{attribute 'GeneratedUsingTerminal: EPP1322-0001-0017'}
{attribute addProperty BoxType "EPP1322-0001-0017"}
{attribute addProperty Id "A_0021_EPP1332_0001_0016A_0021_EPP1332_0001_0016_6B73DC91322"}
{attribute addProperty CRC "3986008381"}
{attribute addProperty Size "322"}
TYPE A_0020_EPP1322_0001_0017_ED95A93D EXTENDS EPP1322_1FC0878B :
STRUCT
	{attribute addProperty Name "A_0021_EPP1332_0001_0016"}
	{attribute addProperty PreviousPort "A_0020(EPP1322-0001-0017) : D"}
	A_0021_EPP1332_0001_0016 : A_0021_EPP1332_0001_0016_6B73DC91;
END_STRUCT
END_TYPE

(* stored: Version 1.2.0.0, ProductVersion 3.1.4024.9
   DUT A_0020_EPP1322_0001_0017_ED95A93D: Id {513a7b3a-4e62-4ca5-a087-986425166cb5} *)
